{attribute addProperty BoxType "EL4712--0000"}
{attribute addProperty Id "Ch1_ValueAT %Q*INT162"}
{attribute addProperty CRC "1318323830"}
{attribute addProperty SizeInBites "16"}
{attribute addProperty SizeInBytes "2"}
TYPE Ch1_Sample_4E940676 :
STRUCT
	{attribute addProperty Name "Ch1_Value"}
	Ch1_Value AT %Q* : INT;
END_STRUCT
END_TYPE

(* stored: Version 1.2.0.0, ProductVersion 3.1.4024.9
   DUT Ch1_Sample_4E940676: Id {7eaee48b-51c7-49c5-8092-ea5035c07cd1} *)
